{attribute 'linkalways'} 
{attribute 'no_explicit_call' := 'This FB is a CLASS and must be accessed using methods or properties'}
{attribute 'enable_dynamic_creation'}
FUNCTION_BLOCK Node_F_VN_ApplyScalingToAffineTransformation EXTENDS VisionNode
VAR
    aTransformationMatrix : _TcVnMatrix2x3_LREAL;
    fScaleX : _LREAL(0.0);
    fScaleY : _LREAL(0.0);
    hrPrev : _HRESULT(S_OK);
	hresult : _HRESULT(S_OK);
END_VAR

METHOD PUBLIC  Clone : I_Node
VAR
	pNode : POINTER TO Node_F_VN_ApplyScalingToAffineTransformation;
END_VAR
pNode := __NEW(Node_F_VN_ApplyScalingToAffineTransformation);
Clone := pNode^;
END_METHOD

METHOD FB_init : BOOL
VAR_INPUT
	bInitRetains : BOOL; // if TRUE, the retain variables are initialized (warm start / cold start)
	bInCopyCode : BOOL;  // if TRUE, the instance afterwards gets moved into the copy code (online change)
END_VAR
AddInput('aTransformationMatrix', aTransformationMatrix);
AddParameter('fScaleX', fScaleX);
AddParameter('fScaleY', fScaleY);
AddInput('hrPrev', hrPrev);
AddOutput('aTransformationMatrix', aTransformationMatrix);
AddOutput('hresult',hresult);
END_METHOD

METHOD PROTECTED  OnExecute : HRESULT
hresult.Value := F_VN_ApplyScalingToAffineTransformation(
	aTransformationMatrix := aTransformationMatrix.Value,
    fScaleX := fScaleX.Value,
    fScaleY := fScaleY.Value,
	hrPrev := hrPrev.Value);
END_METHOD

METHOD PUBLIC PreExecutionCheck
VAR_INPUT
	Check : I_PreExecutionChecks;
END_VAR
END_METHOD

END_FUNCTION_BLOCK

(* stored: Version 1.1.0.1, ProductVersion 3.1.4024.13
   POU Node_F_VN_ApplyScalingToAffineTransformation: Id {a88d640d-c6c0-06da-3e8b-aa98dc673dab}, SpecialFunc None
   Folder Constructor: Id {ac0bf1b0-e33e-06cd-32c7-0e03200a82dd}
   Method Clone: Id {e122a17c-d71e-0387-332a-e1a5e77b3267}
   Method FB_init: Id {e9810eff-20dd-0ebc-26d9-eb0e07f8a265}
   Method OnExecute: Id {0a480762-ecd7-0f14-0ed7-f563d8c80a20}
   Method PreExecutionCheck: Id {de7d2409-86bf-07bc-0c16-9594ff740a34} *)
